// TIA Portal V20 export
TYPE "zp_CITI_Configuration"
// stored: Access Published, Namespace CITI_Logic
   STRUCT
      Instance : DInt;
      UpdatePriority : DInt;
      Features : "CITI_Logic.zp_CITI_Features";
      Parameters { S7_SetPoint := 'True'} : "CITI_Logic.zp_CITI_Parameters";
   END_STRUCT;
END_TYPE
